// TIA Portal V15.1 export
// export: Created 2020-06-12T07:35:47.0068359Z, ExportSetting None, DisplayName Totally Integrated Automation Portal, DisplayVersion V15.1, DisplayName TIA Portal Openness, DisplayVersion V15.1, DisplayName STEP 7 Professional, DisplayVersion V15.1, DisplayName STEP 7 Safety, DisplayVersion V15.1, DisplayName WinCC Advanced, DisplayVersion V15.1
FUNCTION "ELC_weight" : Void   // FC80, FBD
TITLE = Elcectrode Movement Control
{ S7_Optimized_Access := 'FALSE' }
// #_contr_up
// #_contr_dwn
// stored: SetENOAutomatically False
   VAR_TEMP
      _csf : Bool;
      _man : Bool;
      _fl_auto_up : Bool;
      _td_pos_fst : Real;
      _clc_end : Real;
      tSetTara : Bool;
      tMaxCnsWeight : Real;
      _netto : Real;
      tAthmoPress : Real;
      tHoodCrossArea : Real;
      tAddedWeight : Real;
      tReqSetTara : Bool;
      tMaxOvlWeight : Real;
      tMaxLimWeight : Real;
      tCompWeight : Real;
   END_VAR
   VAR_TEMP   // added for the SCL form of the ladder/FBD networks
      _w1 : Bool;
   END_VAR
BEGIN

REGION Network 1: Set Zero
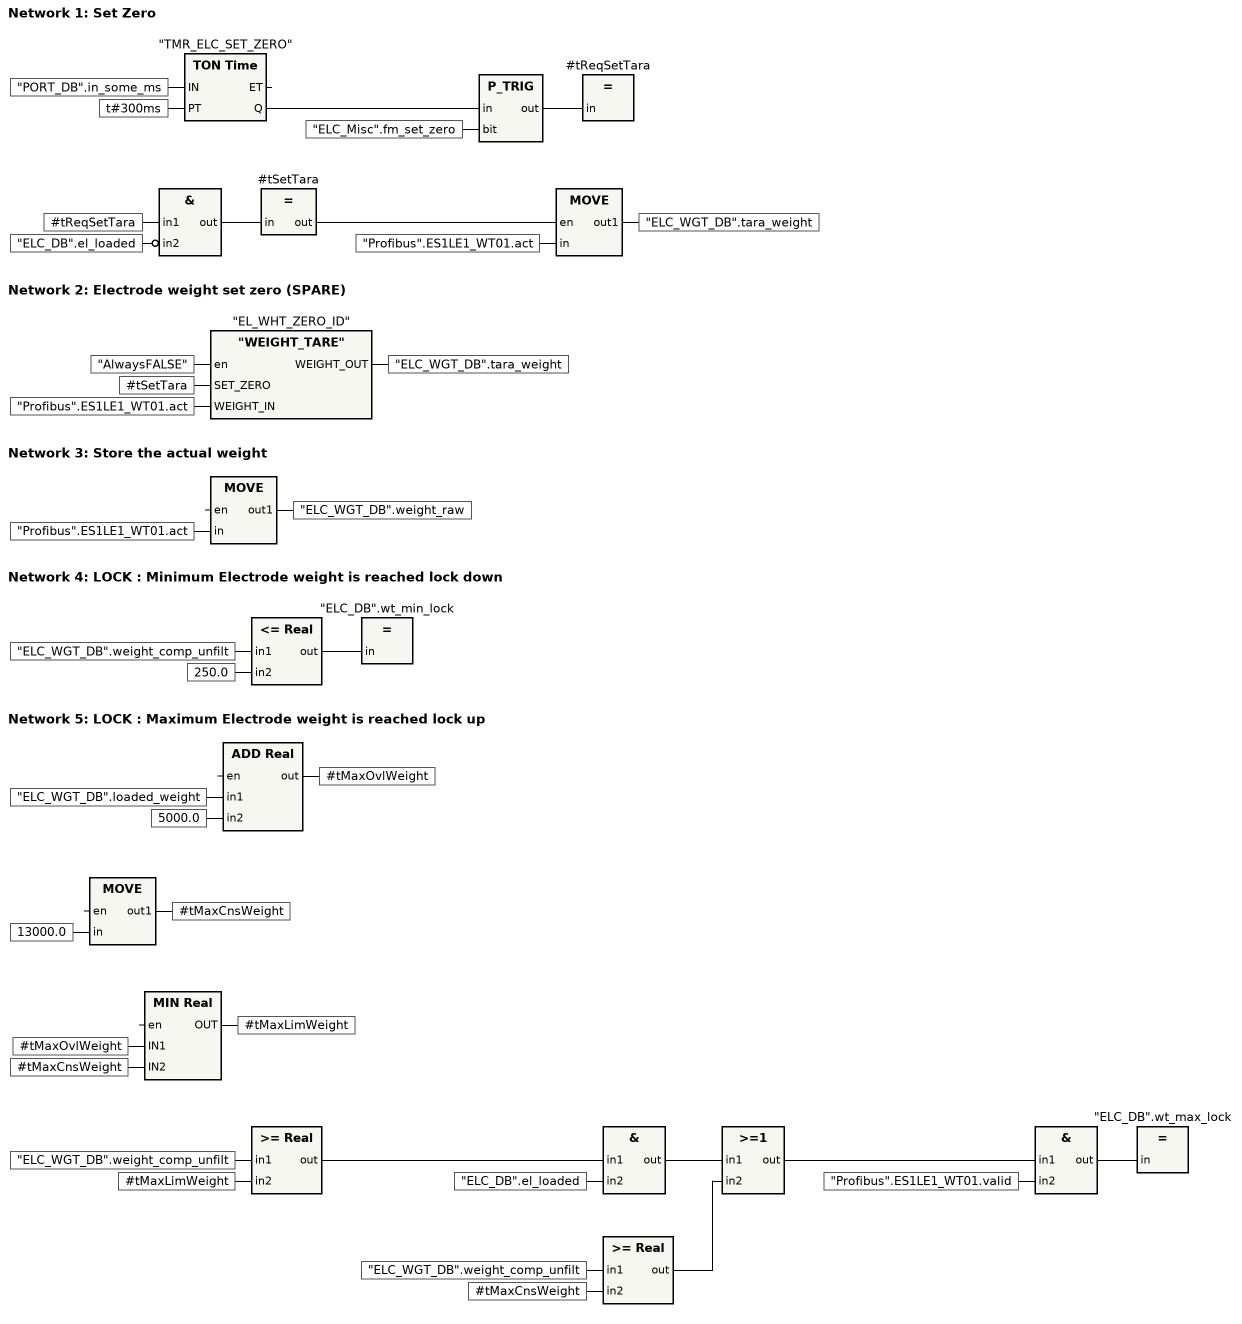
   "TMR_ELC_SET_ZERO".TON(IN := "PORT_DB".in_some_ms, PT := t#300ms);
   #_w1 := "TMR_ELC_SET_ZERO".Q AND NOT "ELC_Misc".fm_set_zero;   // rising edge
   "ELC_Misc".fm_set_zero := "TMR_ELC_SET_ZERO".Q;
   #tReqSetTara := #_w1;
   #tSetTara := #tReqSetTara AND NOT "ELC_DB".el_loaded;
   IF #tSetTara THEN "ELC_WGT_DB".tara_weight := "Profibus".ES1LE1_WT01.act; END_IF;
END_REGION

REGION Network 2: Electrode weight set zero (SPARE)
   // VLS: problem after PLC restart
   IF "AlwaysFALSE" THEN
       "EL_WHT_ZERO_ID"(SET_ZERO := #tSetTara,   // "WEIGHT_TARE"
                        WEIGHT_IN := "Profibus".ES1LE1_WT01.act,
                        WEIGHT_OUT => "ELC_WGT_DB".tara_weight);
   END_IF;
END_REGION

REGION Network 3: Store the actual weight
   "ELC_WGT_DB".weight_raw := "Profibus".ES1LE1_WT01.act;
END_REGION

REGION Network 4: LOCK : Minimum Electrode weight is reached lock down
   "ELC_DB".wt_min_lock := "ELC_WGT_DB".weight_comp_unfilt <= 250.0;
END_REGION

REGION Network 5: LOCK : Maximum Electrode weight is reached lock up
   #tMaxOvlWeight := "ELC_WGT_DB".loaded_weight + 5000.0;
   #tMaxCnsWeight := 13000.0;
   #tMaxLimWeight := MIN(IN1 := #tMaxOvlWeight, IN2 := #tMaxCnsWeight);
   "ELC_DB".wt_max_lock := ((("ELC_WGT_DB".weight_comp_unfilt >= #tMaxLimWeight) AND "ELC_DB".el_loaded) OR ("ELC_WGT_DB".weight_comp_unfilt >= #tMaxCnsWeight)) AND "Profibus".ES1LE1_WT01.valid;
END_REGION

REGION Network 6: Electrode is catched
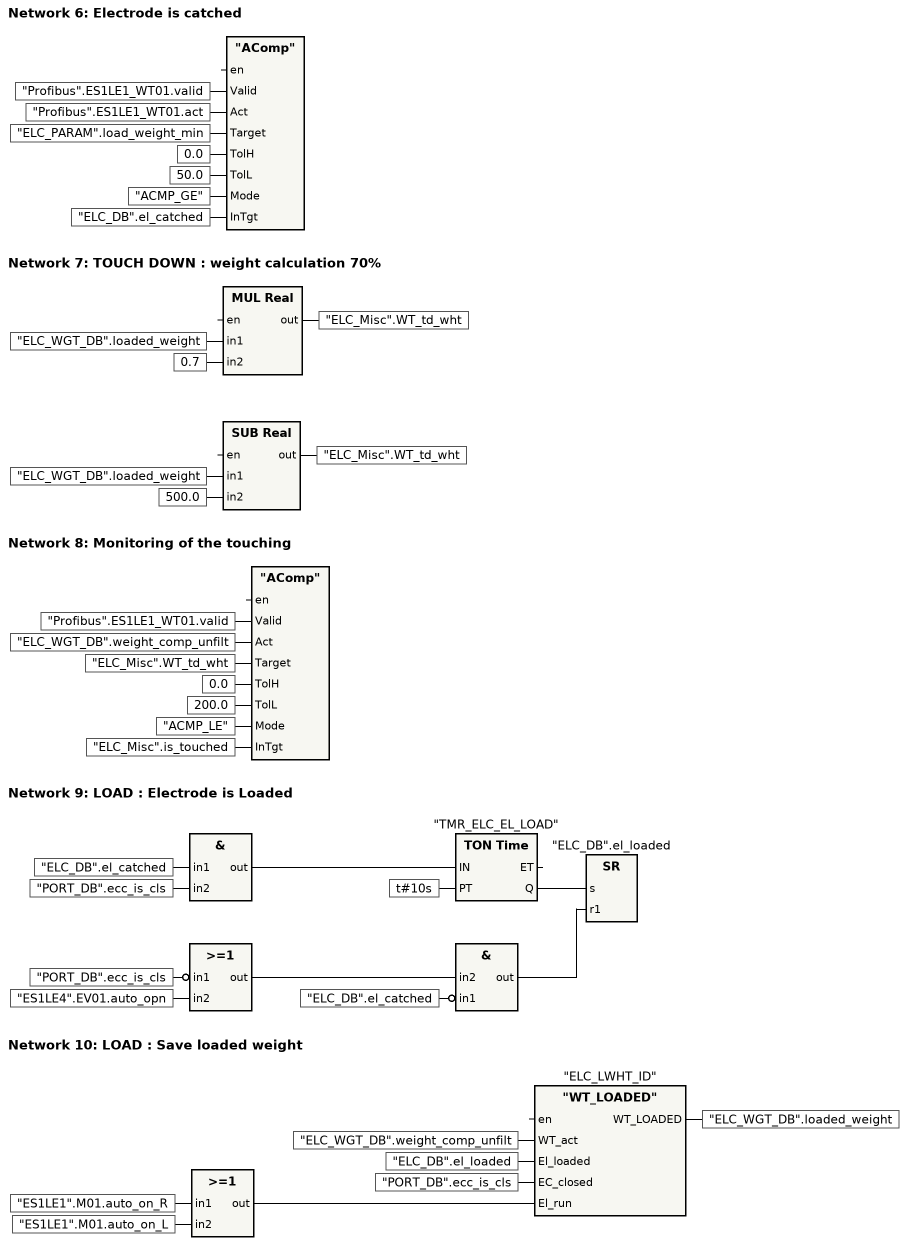
   "AComp"(Valid := "Profibus".ES1LE1_WT01.valid,
           Act := "Profibus".ES1LE1_WT01.act,
           Target := "ELC_PARAM".load_weight_min,
           TolH := 0.0,
           TolL := 50.0,
           Mode := "ACMP_GE",
           InTgt := "ELC_DB".el_catched);
END_REGION

REGION Network 7: TOUCH DOWN : weight calculation 70%
   "ELC_Misc".WT_td_wht := "ELC_WGT_DB".loaded_weight * 0.7;
   "ELC_Misc".WT_td_wht := "ELC_WGT_DB".loaded_weight - 500.0;
END_REGION

REGION Network 8: Monitoring of the touching
   "AComp"(Valid := "Profibus".ES1LE1_WT01.valid,
           Act := "ELC_WGT_DB".weight_comp_unfilt,
           Target := "ELC_Misc".WT_td_wht,
           TolH := 0.0,
           TolL := 200.0,
           Mode := "ACMP_LE",
           InTgt := "ELC_Misc".is_touched);
END_REGION

REGION Network 9: LOAD : Electrode is Loaded
   // Set:
   // - Electrode WT >= WT_loaded
   // - Electrode clamp is closed
   // 
   // Reset:
   // - Electrode WT < WT_loaded
   // - Electrode clamp is opened
   // - ELWA in unload position
   "TMR_ELC_EL_LOAD".TON(IN := "ELC_DB".el_catched AND "PORT_DB".ecc_is_cls, PT := t#10s);
   IF "TMR_ELC_EL_LOAD".Q THEN
       "ELC_DB".el_loaded := TRUE;   // SR flip-flop
   END_IF;
   IF (NOT "PORT_DB".ecc_is_cls OR "ES1LE4".EV01.auto_opn) AND NOT "ELC_DB".el_catched THEN
       "ELC_DB".el_loaded := FALSE;
   END_IF;
END_REGION

REGION Network 10: LOAD : Save loaded weight
   "ELC_LWHT_ID"(WT_act := "ELC_WGT_DB".weight_comp_unfilt,   // "WT_LOADED"
                 El_loaded := "ELC_DB".el_loaded,
                 EC_closed := "PORT_DB".ecc_is_cls,
                 El_run := "ES1LE1".M01.auto_on_R OR "ES1LE1".M01.auto_on_L,
                 WT_LOADED => "ELC_WGT_DB".loaded_weight);
END_REGION

REGION Network 11: ** NEW **
END_REGION

REGION Network 12: Average signal of WT01 electode weight, kg
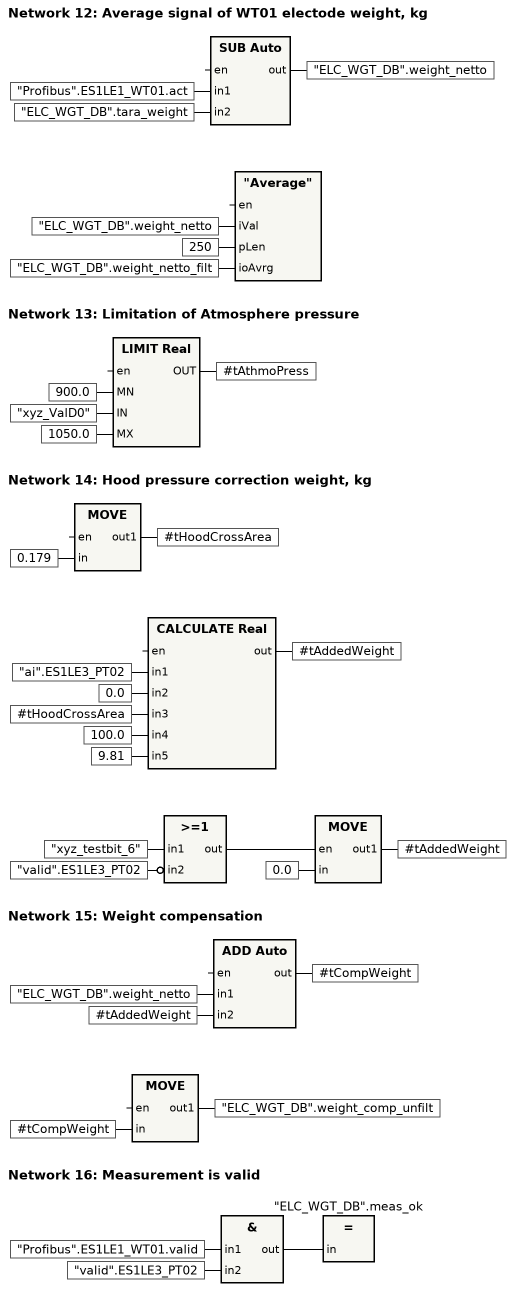
   "ELC_WGT_DB".weight_netto := "Profibus".ES1LE1_WT01.act - "ELC_WGT_DB".tara_weight;
   "Average"(iVal := "ELC_WGT_DB".weight_netto, pLen := 250, ioAvrg := "ELC_WGT_DB".weight_netto_filt);
END_REGION

REGION Network 13: Limitation of Atmosphere pressure
   // "ai".ES1LZ1_PT01
   #tAthmoPress := LIMIT(MN := 900.0, IN := "xyz_ValD0", MX := 1050.0);
END_REGION

REGION Network 14: Hood pressure correction weight, kg
   // Hood WST = 0.178
   // Hood Uddeholm = 0.257
   // 
   // PuM: I disabled this because there is not DPT or athmosperic pressure measuremnt
   #tHoodCrossArea := 0.179;
   #tAddedWeight := ("ai".ES1LE3_PT02-0.0)*#tHoodCrossArea*100.0/9.81;
   IF "xyz_testbit_6" OR NOT "valid".ES1LE3_PT02 THEN #tAddedWeight := 0.0; END_IF;
END_REGION

REGION Network 15: Weight compensation
   #tCompWeight := "ELC_WGT_DB".weight_netto + #tAddedWeight;
   "ELC_WGT_DB".weight_comp_unfilt := #tCompWeight;
END_REGION

REGION Network 16: Measurement is valid
   "ELC_WGT_DB".meas_ok := "Profibus".ES1LE1_WT01.valid AND "valid".ES1LE3_PT02;
END_REGION

REGION Network 17: Average signal of hood pressure correction weight, kg
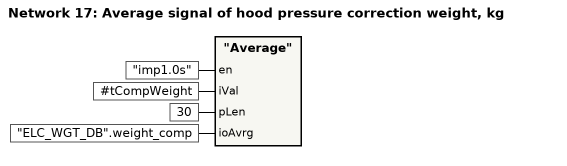
   IF "imp1.0s" THEN "Average"(iVal := #tCompWeight, pLen := 30, ioAvrg := "ELC_WGT_DB".weight_comp); END_IF;
END_REGION
END_FUNCTION
